(* Logix 5000 project; controller ESP_300kVA_L24ERM vendor 1 type 14 code 150 rev 33.12; software revision 33.01 *)

TASK MainTask (continuous, watchdog 500 ms) : MainProgram

MODULES
   Local : vendor 1 type 14 code 150 (Compact 0, rev 33.12)
      Discrete_IO : Embedded (Compact 1, rev 3.1, Output RPI 20 ms)
      Counters : Embedded (Compact 3, rev 1.1, Output RPI 20 ms)
      Analog_IO : Embedded (Compact 2, rev 1.1, Output RPI 80 ms)
      PowerFlex755PMM : vendor 1 type 143 code 6288 (Ethernet 192.168.2.160, rev 3.2, Output RPI 20 ms)
           PowerFlex755PMM:O.P14_DLXDINTInSP1   // Bit de Falla General
          : vendor 1 type 143 code 33184 (RhinoBP 14, rev 2.5)
          : vendor 1 type 143 code 32928 (RhinoBP 13, rev 1.1)
          : vendor 1 type 143 code 767 (RhinoBP 1, rev 2.7)
          : vendor 1 type 143 code 416 (RhinoBP 6, rev 1.8)
          : vendor 1 type 143 code 416 (RhinoBP 4, rev 1.8)
          : vendor 1 type 143 code 416 (RhinoBP 5, rev 1.8)
          : vendor 1 type 143 code 24736 (RhinoBP 7, rev 1.1)
      PowerFlex755IM : PowerFlex 755-EENET (Ethernet 192.168.2.10, rev 14.5, Output RPI 20 ms)
          : vendor 1 type 143 code 416 (RhinoBP 4, rev 1.8)
          : vendor 1 type 143 code 24736 (RhinoBP 7, rev 1.1)
          : vendor 1 type 143 code 416 (RhinoBP 5, rev 1.8)
          : vendor 1 type 143 code 767 (RhinoBP 1, rev 2.7)
          : vendor 1 type 143 code 32928 (RhinoBP 13, rev 1.1)
          : vendor 1 type 143 code 33184 (RhinoBP 14, rev 2.5)
          : vendor 1 type 143 code 416 (RhinoBP 6, rev 1.8)
END_MODULES

TYPE DIO_Fn :   // UDT Para Canales
STRUCT
   Channel : INT;   // Número del canal
   Type : BOOL;   // Typo de entrada (0:NO,1:NC) Tipo de salida (0:HA,1LA)
   Value : BOOL;   // Valor de la función
   Enable : BOOL;   // Habilitador
END_STRUCT
END_TYPE

TYPE Protecciones :
STRUCT
   Enable_HH : BOOL[32];   // Disparo por alto alto habilitado
   SetPoint_HH : REAL[32];   // Límite disparo HH
   TripTime_HH : INT[32];   // Tiempo disparo HH
   Enable_LL : BOOL[32];   // Disparo por bajo bajo habilitado
   SetPoint_LL : REAL[32];   // Límite disparo LL
   TripTime_LL : INT[32];   // Tiempo disparo LL
   Disparo_HH : BOOL[32];   // Estado de la señal de disparo HH
   Disparo_LL : BOOL[32];   // Estado de la señal de disparo LL
   Type : INT;   // Tipo de Protección
END_STRUCT
END_TYPE

ADD_ON_INSTRUCTION BMUX_16_1   (* revision 0.1 *)
// 16:1 BOOL MUX
VAR_INPUT
   INPUT : INT; {visible}   // Entrada
   SEL : INT; {visible}   // Selector
END_VAR
VAR_OUTPUT
   OUT : BOOL; {access Read Only, visible}   // Salida
END_VAR
VAR_INPUT
   TYPE : BOOL;
END_VAR
VAR
   MUX_8_1_01 : BMUX_8_1; {access None}
   MUX_8_1_02 : BMUX_8_1; {access None}
   BAND_01 : FBD_BOOLEAN_AND := (In1 := 1, In2 := 1, In3 := 1, In4 := 1, In5 := 1, In6 := 1, In7 := 1, In8 := 1); {access None}
   BAND_02 : FBD_BOOLEAN_AND := (In1 := 1, In2 := 1, In3 := 1, In4 := 1, In5 := 1, In6 := 1, In7 := 1, In8 := 1); {access None}
   BNOT_01 : FBD_BOOLEAN_NOT := (In := 1); {access None}
   BOR_01 : FBD_BOOLEAN_OR; {access None}
   __l13611DCB8D0E7587 : INT; {access None}
   __lD1E1ECCF935F20E9 : INT; {access None}
   __lCDF1D212B6E33786 : BOOL; {access None}
END_VAR

ROUTINE Logic   (* function block diagram *)
   SHEET 1
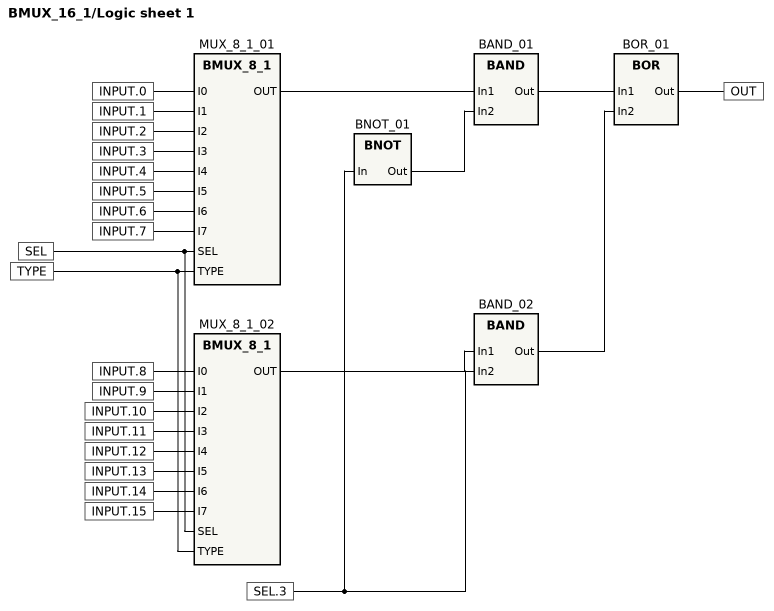
   MUX_8_1_01 : BMUX_8_1(I0 := INPUT.0, I1 := INPUT.1, I2 := INPUT.2, I3 := INPUT.3, I4 := INPUT.4, I5 := INPUT.5, I6 := INPUT.6, I7 := INPUT.7, SEL := SEL, TYPE := TYPE);
   MUX_8_1_02 : BMUX_8_1(I0 := INPUT.8, I1 := INPUT.9, I2 := INPUT.10, I3 := INPUT.11, I4 := INPUT.12, I5 := INPUT.13, I6 := INPUT.14, I7 := INPUT.15, SEL := SEL, TYPE := TYPE);
   BNOT_01 : BNOT(In := SEL.3);
   BAND_01 : BAND(In1 := MUX_8_1_01.OUT, In2 := BNOT_01.Out);
   BAND_02 : BAND(In1 := MUX_8_1_02.OUT, In2 := SEL.3);
   BOR_01 : BOR(In1 := BAND_01.Out, In2 := BAND_02.Out);
   OUT := BOR_01.Out;
END_ROUTINE
END_ADD_ON_INSTRUCTION

ADD_ON_INSTRUCTION BMUX_4_1   (* revision 0.1 *)
// 4:1 BOOL MUX
VAR_INPUT
   I0 : BOOL; {visible}   // Entrada 0
   I1 : BOOL; {visible}   // Entrada 1
   I2 : BOOL; {visible}   // Entrada 2
   I3 : BOOL; {visible}   // Entrada 3
   SEL : INT; {visible}   // Selector
END_VAR
VAR_OUTPUT
   OUT : BOOL; {visible}   // Salida
END_VAR
VAR_INPUT
   TYPE : BOOL;
END_VAR
VAR
   BAND_01 : FBD_BOOLEAN_AND := (In1 := 1, In2 := 1, In3 := 1, In4 := 1, In5 := 1, In6 := 1, In7 := 1, In8 := 1); {access None}
   BAND_02 : FBD_BOOLEAN_AND := (In1 := 1, In2 := 1, In3 := 1, In4 := 1, In5 := 1, In6 := 1, In7 := 1, In8 := 1); {access None}
   BAND_03 : FBD_BOOLEAN_AND := (In1 := 1, In2 := 1, In3 := 1, In4 := 1, In5 := 1, In6 := 1, In7 := 1, In8 := 1); {access None}
   BAND_04 : FBD_BOOLEAN_AND := (In1 := 1, In2 := 1, In3 := 1, In4 := 1, In5 := 1, In6 := 1, In7 := 1, In8 := 1); {access None}
   BOR_01 : FBD_BOOLEAN_OR; {access None}
   BNOT_01 : FBD_BOOLEAN_NOT := (In := 1); {access None}
   BNOT_02 : FBD_BOOLEAN_NOT := (In := 1); {access None}
   BAND_05 : FBD_BOOLEAN_AND := (In1 := 1, In2 := 1, In3 := 1, In4 := 1, In5 := 1, In6 := 1, In7 := 1, In8 := 1);
   BAND_06 : FBD_BOOLEAN_AND := (In1 := 1, In2 := 1, In3 := 1, In4 := 1, In5 := 1, In6 := 1, In7 := 1, In8 := 1);
   BNOT_03 : FBD_BOOLEAN_NOT := (In := 1);
   BNOT_04 : FBD_BOOLEAN_NOT := (In := 1);
   BOR_02 : FBD_BOOLEAN_OR;
   __lA34AA79BD695A9B9 : INT; {access None}
   __l3F476DF96765899A : BOOL; {access None}
   __lA5B7ACC4E5B37ACF : BOOL; {access None}
   __l435C749CB0444308 : BOOL; {access None}
   __lD1FFE671015823D2 : BOOL; {access None}
   __l62043FB7EA6F2954 : BOOL; {access None}
END_VAR

ROUTINE Logic   (* function block diagram *)
   SHEET 1
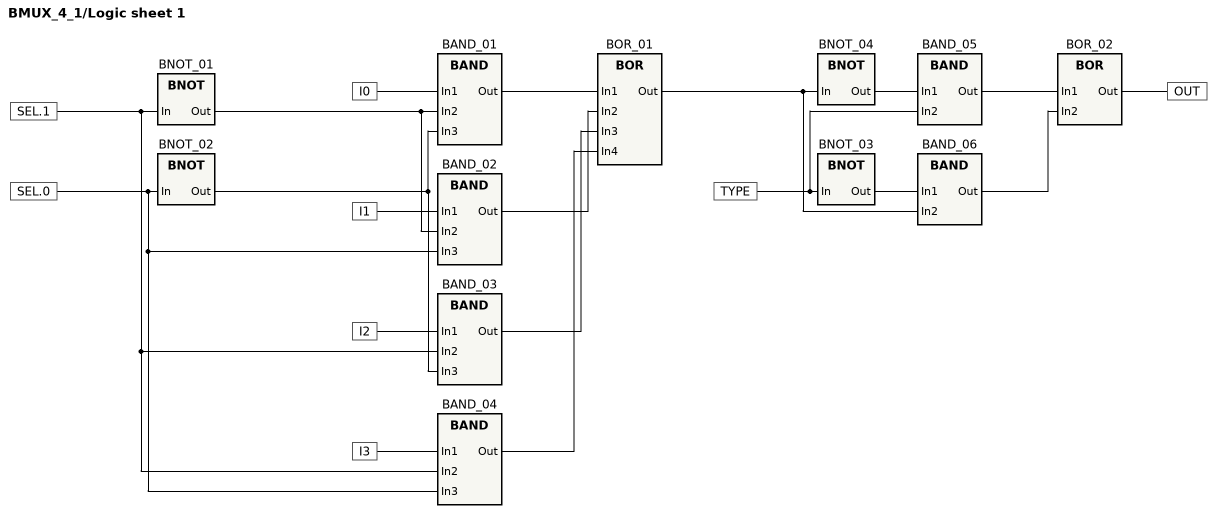
   BNOT_01 : BNOT(In := SEL.1);
   BNOT_02 : BNOT(In := SEL.0);
   BAND_01 : BAND(In1 := I0, In2 := BNOT_01.Out, In3 := BNOT_02.Out);
   BAND_02 : BAND(In1 := I1, In2 := BNOT_01.Out, In3 := SEL.0);
   BAND_03 : BAND(In1 := I2, In2 := SEL.1, In3 := BNOT_02.Out);
   BAND_04 : BAND(In1 := I3, In2 := SEL.1, In3 := SEL.0);
   BOR_01 : BOR(In1 := BAND_01.Out, In2 := BAND_02.Out, In3 := BAND_03.Out, In4 := BAND_04.Out);
   BNOT_04 : BNOT(In := BOR_01.Out);
   BNOT_03 : BNOT(In := TYPE);
   BAND_05 : BAND(In1 := BNOT_04.Out, In2 := TYPE);
   BAND_06 : BAND(In1 := BNOT_03.Out, In2 := BOR_01.Out);
   BOR_02 : BOR(In1 := BAND_05.Out, In2 := BAND_06.Out);
   OUT := BOR_02.Out;
END_ROUTINE
END_ADD_ON_INSTRUCTION

ADD_ON_INSTRUCTION BMUX_8_1   (* revision 0.1 *)
// 8:1 BOOL MUX
VAR_INPUT
   I0 : BOOL; {visible}   // Entrada 0
   I1 : BOOL; {visible}   // Entrada 1
   I2 : BOOL; {visible}   // Entrada 2
   I3 : BOOL; {visible}   // Entrada 3
   I4 : BOOL; {visible}   // Entrada 4
   I5 : BOOL; {visible}   // Entrada 5
   I6 : BOOL; {visible}   // Entrada 6
   I7 : BOOL; {visible}   // Entrada 7
   SEL : INT; {visible}   // Selector
END_VAR
VAR_OUTPUT
   OUT : BOOL; {visible}   // Salida
END_VAR
VAR_INPUT
   TYPE : BOOL;
END_VAR
VAR
   BAND_01 : FBD_BOOLEAN_AND := (In1 := 1, In2 := 1, In3 := 1, In4 := 1, In5 := 1, In6 := 1, In7 := 1, In8 := 1); {access None}
   BAND_02 : FBD_BOOLEAN_AND := (In1 := 1, In2 := 1, In3 := 1, In4 := 1, In5 := 1, In6 := 1, In7 := 1, In8 := 1); {access None}
   MUX_4_1_02 : BMUX_4_1; {access None}
   MUX_4_1_01 : BMUX_4_1; {access None}
   BNOT_01 : FBD_BOOLEAN_NOT := (In := 1); {access None}
   BOR_01 : FBD_BOOLEAN_OR; {access None}
   __l3844A21951326208 : INT; {access None}
   __l92E31AA3E07A0FB5 : BOOL; {access None}
   __lFC38970C7D342C75 : BOOL; {access None}
   __l740E29C8E41AD4FE : BOOL; {access None}
   __l47807FE8D131736A : BOOL; {access None}
   __lC8897F2B9FAED5C5 : BOOL; {access None}
   __lCFCD8E0D59ED18C9 : BOOL; {access None}
   __l6FFFD8D902218155 : BOOL; {access None}
   __lC2B98392E907BE62 : BOOL; {access None}
   __l3C983B185907781A : BOOL; {access None}
END_VAR

ROUTINE Logic   (* function block diagram *)
   SHEET 1
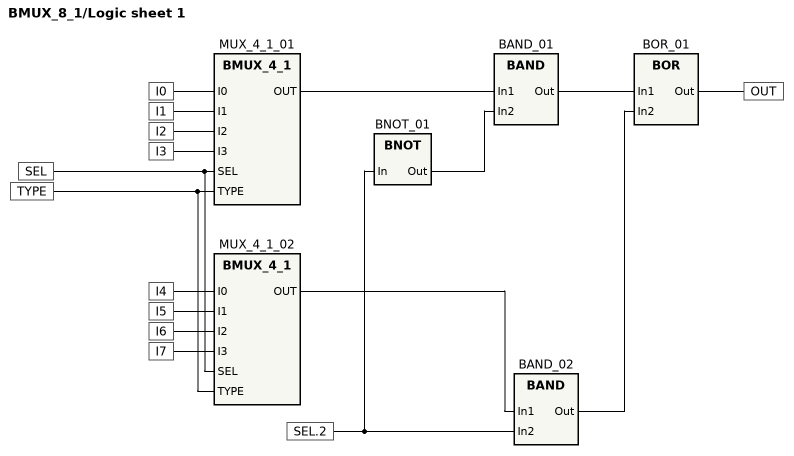
   MUX_4_1_01 : BMUX_4_1(I0 := I0, I1 := I1, I2 := I2, I3 := I3, SEL := SEL, TYPE := TYPE);
   MUX_4_1_02 : BMUX_4_1(I0 := I4, I1 := I5, I2 := I6, I3 := I7, SEL := SEL, TYPE := TYPE);
   BNOT_01 : BNOT(In := SEL.2);
   BAND_01 : BAND(In1 := MUX_4_1_01.OUT, In2 := BNOT_01.Out);
   BAND_02 : BAND(In1 := MUX_4_1_02.OUT, In2 := SEL.2);
   BOR_01 : BOR(In1 := BAND_01.Out, In2 := BAND_02.Out);
   OUT := BOR_01.Out;
END_ROUTINE
END_ADD_ON_INSTRUCTION

VAR_GLOBAL   (* controller tags *)
   ChannelSel : INT[16];
   DOChannel : INT;
   Falla_general : BOOL;
   Filtro_armonicos : BOOL;
   Reset : BOOL;
   VSD_BitFalla : DINT;
END_VAR

PROGRAM MainProgram   (* main routine MainRoutine *)
VAR
   BMUX_16_1_01 : BMUX_16_1 := (INPUT := 1743);
   BMUX_16_1_02 : BMUX_16_1 := (INPUT := 1743);
   BMUX_16_1_03 : BMUX_16_1 := (INPUT := 1743);
   BMUX_16_1_04 : BMUX_16_1 := (INPUT := 1743, TYPE := 1);
   BMUX_16_1_05 : BMUX_16_1 := (INPUT := 1743);
   BMUX_16_1_06 : BMUX_16_1 := (INPUT := 1743, SEL := 5);
   BMUX_16_1_07 : BMUX_16_1 := (INPUT := 1743, SEL := 4);
   BMUX_16_1_08 : BMUX_16_1 := (INPUT := 1743, SEL := 2, TYPE := 1);
   BMUX_16_1_09 : BMUX_16_1 := (INPUT := 1743, SEL := 3, TYPE := 1);
   BMUX_16_1_10 : BMUX_16_1 := (INPUT := 1743, SEL := 6, TYPE := 1);
   BMUX_16_1_11 : BMUX_16_1 := (INPUT := 1743, SEL := 7, TYPE := 1);
   BMUX_16_1_12 : BMUX_16_1 := (INPUT := 1743, SEL := 1, TYPE := 1);
   BMUX_16_1_13 : BMUX_16_1 := (INPUT := 1743);
   BMUX_16_1_14 : BMUX_16_1 := (INPUT := 1743);
   BMUX_16_1_15 : BMUX_16_1 := (INPUT := 1743, TYPE := 1);
   BMUX_16_1_16 : BMUX_16_1 := (INPUT := 1743);
   BMUX_16_1_17 : BMUX_16_1 := (INPUT := 1743);
   BMUX_16_1_18 : BMUX_16_1 := (INPUT := 1743, SEL := 8);
   BMUX_16_1_19 : BMUX_16_1;
   BMUX_4_1_02 : BMUX_4_1 := (SEL := 2);
   BMUX_4_1_03 : BMUX_4_1 := (SEL := 3);
   BMUX_4_1_04 : BMUX_4_1 := (SEL := 1);
   BMUX_4_1_05 : BMUX_4_1;
   BMUX_4_1_06 : BMUX_4_1;
   BMUX_4_1_07 : BMUX_4_1;
   BMUX_4_1_08 : BMUX_4_1;
   BMUX_4_1_09 : BMUX_4_1;
   BMUX_4_1_10 : BMUX_4_1;
   BMUX_4_1_11 : BMUX_4_1;
   BMUX_4_1_12 : BMUX_4_1;
   BMUX_4_1_13 : BMUX_4_1;
   BMUX_4_1_14 : BMUX_4_1;
   BMUX_4_1_15 : BMUX_4_1;
   BMUX_4_1_16 : BMUX_4_1;
   BMUX_4_1_17 : BMUX_4_1;
   BOR_01 : FBD_BOOLEAN_OR;
   BOR_02 : FBD_BOOLEAN_OR;
   BOR_03 : FBD_BOOLEAN_OR;
   BOR_04 : FBD_BOOLEAN_OR;
   BOR_05 : FBD_BOOLEAN_OR;
   BOR_06 : FBD_BOOLEAN_OR;
   BOR_07 : FBD_BOOLEAN_OR;
   BOR_08 : FBD_BOOLEAN_OR;
   BOR_09 : FBD_BOOLEAN_OR;
   BOR_10 : FBD_BOOLEAN_OR;
   BOR_11 : FBD_BOOLEAN_OR;
   BOR_12 : FBD_BOOLEAN_OR;
   BOR_13 : FBD_BOOLEAN_OR;
   BOR_14 : FBD_BOOLEAN_OR;
   BOR_15 : FBD_BOOLEAN_OR;
   BOR_16 : FBD_BOOLEAN_OR;
   BOR_17 : FBD_BOOLEAN_OR;
   BOR_18 : FBD_BOOLEAN_OR;
   BOR_19 : FBD_BOOLEAN_OR;
   BXOR_01 : FBD_BOOLEAN_XOR;
   DI_Alarma_alta_temperatura_SUT : DIO_Fn := (Channel := 4, Enable := 1);
   DI_Alarma_bajo_nivel_aceite_SUT : DIO_Fn := (Channel := 2, Type := 1, Enable := 1);
   DI_Alarma_DPS : DIO_Fn := (Channel := 7, Type := 1, Enable := 1);
   DI_Disparo_alta_presion_THP : DIO_Fn;
   DI_Disparo_alta_temperatura_filtros : DIO_Fn := (Channel := 1, Type := 1, Enable := 1);
   DI_Disparo_alta_temperatura_SUT : DIO_Fn := (Channel := 5, Enable := 1);
   DI_Disparo_alto_nivel_aceite_SUT : DIO_Fn;
   DI_Disparo_baja_presion_troncal : DIO_Fn;
   DI_Disparo_bajo_bajo_nivel_aceite_SUT : DIO_Fn := (Channel := 3, Type := 1, Enable := 1);
   DI_Disparo_puerta_abierta : DIO_Fn;
   DI_Disparo_shutdown_SCC : DIO_Fn := (Channel := 8, Enable := 1);
   DI_Disparo_sobre_tension_SUT : DIO_Fn;
   DI_Disparo_valvula_sobrepresion_SUT : DIO_Fn := (Channel := 6, Type := 1, Enable := 1);
   DI_Proteccion_termica_motor : DIO_Fn;
   DI_Reset : DIO_Fn;
   DI_Start : DIO_Fn;
   DI_Stop : DIO_Fn;
   DI_Stop_ESD : DIO_Fn := (Type := 1, Enable := 1);
   DI_Stop_ESD_Remoto : DIO_Fn;
   DO_Disparo_breaker_ESD : DIO_Fn;
   DO_Falla_general : DIO_Fn := (Channel := 2, Value := 1, Enable := 1);
   MUX_01 : MULTIPLEXER := (Status := 16#0000_0003, InstructFault := 1, SelectorInv := 1);
   Protecciones : Protecciones;
   TON_ProteccionHH : TIMER[16];
   TON_ProteccionLL : TIMER[16];
END_VAR

ROUTINE Input_Output   (* function block diagram *)
// Rutina para el control de entradas y salidas Digitales
   SHEET 1   // Funciones de entrada 1
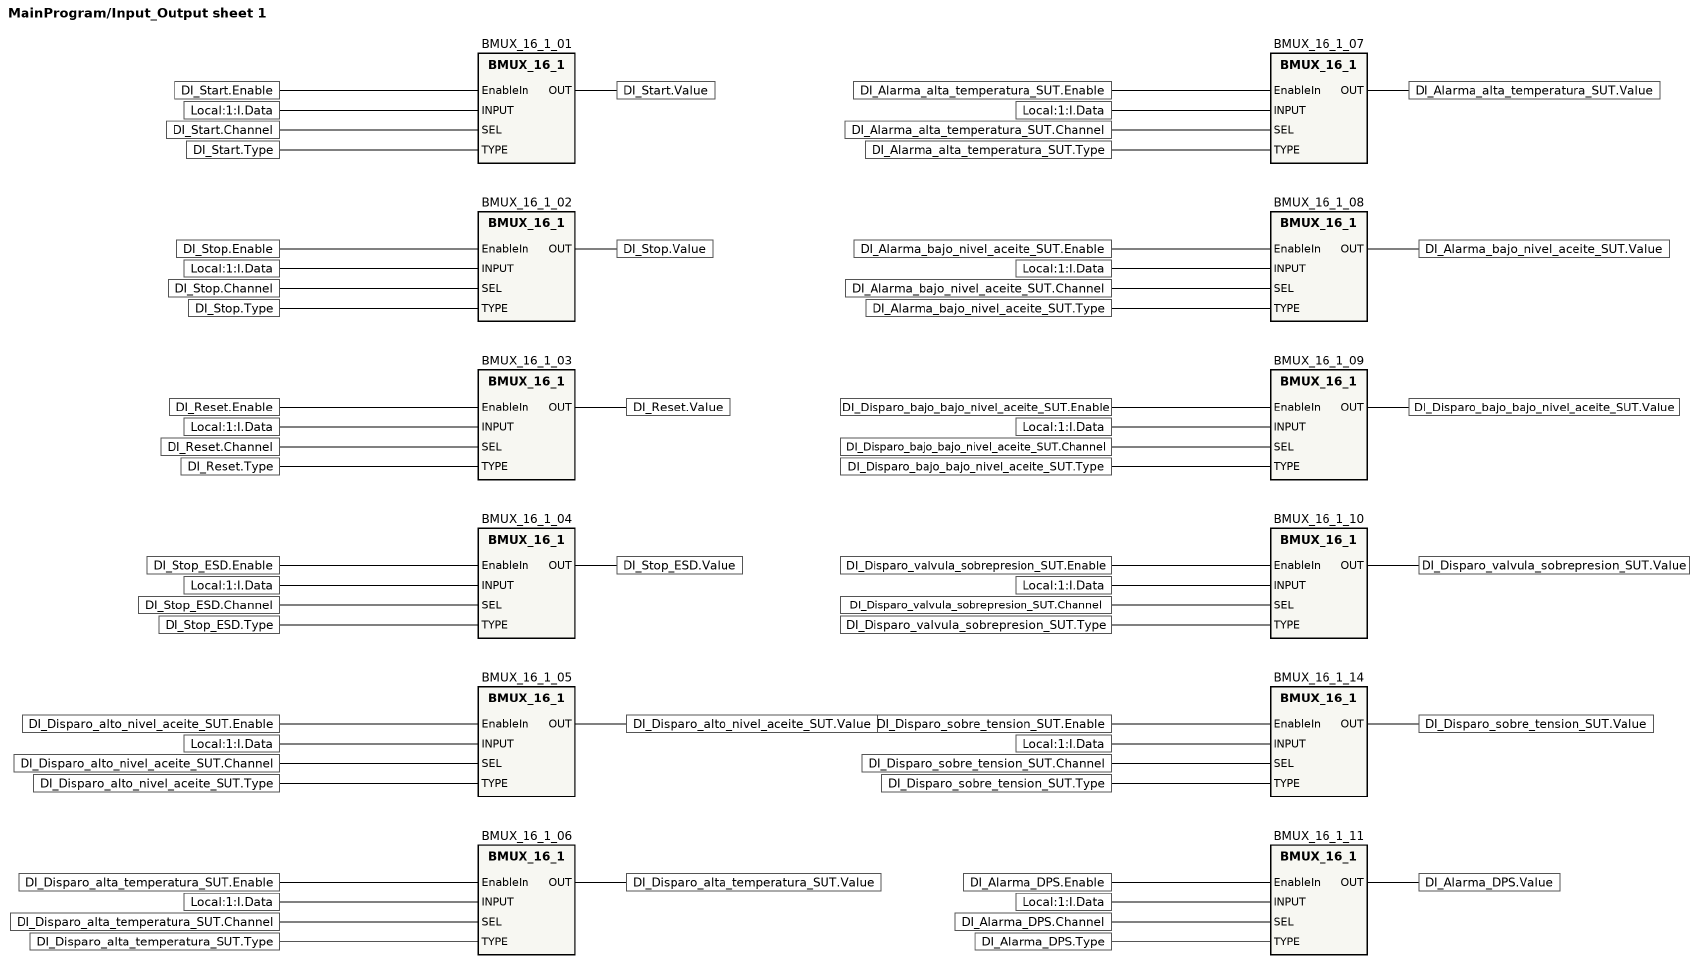
   BMUX_16_1_01 : BMUX_16_1(EnableIn := DI_Start.Enable, INPUT := Local:1:I.Data, SEL := DI_Start.Channel, TYPE := DI_Start.Type);
   BMUX_16_1_02 : BMUX_16_1(EnableIn := DI_Stop.Enable, INPUT := Local:1:I.Data, SEL := DI_Stop.Channel, TYPE := DI_Stop.Type);
   BMUX_16_1_03 : BMUX_16_1(EnableIn := DI_Reset.Enable, INPUT := Local:1:I.Data, SEL := DI_Reset.Channel, TYPE := DI_Reset.Type);
   BMUX_16_1_04 : BMUX_16_1(EnableIn := DI_Stop_ESD.Enable, INPUT := Local:1:I.Data, SEL := DI_Stop_ESD.Channel, TYPE := DI_Stop_ESD.Type);
   BMUX_16_1_05 : BMUX_16_1(EnableIn := DI_Disparo_alto_nivel_aceite_SUT.Enable, INPUT := Local:1:I.Data, SEL := DI_Disparo_alto_nivel_aceite_SUT.Channel, TYPE := DI_Disparo_alto_nivel_aceite_SUT.Type);
   BMUX_16_1_06 : BMUX_16_1(EnableIn := DI_Disparo_alta_temperatura_SUT.Enable, INPUT := Local:1:I.Data, SEL := DI_Disparo_alta_temperatura_SUT.Channel, TYPE := DI_Disparo_alta_temperatura_SUT.Type);
   DI_Start.Value := BMUX_16_1_01.OUT;
   DI_Stop.Value := BMUX_16_1_02.OUT;
   DI_Stop_ESD.Value := BMUX_16_1_04.OUT;
   DI_Reset.Value := BMUX_16_1_03.OUT;
   DI_Disparo_alto_nivel_aceite_SUT.Value := BMUX_16_1_05.OUT;
   DI_Disparo_alta_temperatura_SUT.Value := BMUX_16_1_06.OUT;
   BMUX_16_1_07 : BMUX_16_1(EnableIn := DI_Alarma_alta_temperatura_SUT.Enable, INPUT := Local:1:I.Data, SEL := DI_Alarma_alta_temperatura_SUT.Channel, TYPE := DI_Alarma_alta_temperatura_SUT.Type);
   BMUX_16_1_08 : BMUX_16_1(EnableIn := DI_Alarma_bajo_nivel_aceite_SUT.Enable, INPUT := Local:1:I.Data, SEL := DI_Alarma_bajo_nivel_aceite_SUT.Channel, TYPE := DI_Alarma_bajo_nivel_aceite_SUT.Type);
   BMUX_16_1_09 : BMUX_16_1(EnableIn := DI_Disparo_bajo_bajo_nivel_aceite_SUT.Enable, INPUT := Local:1:I.Data, SEL := DI_Disparo_bajo_bajo_nivel_aceite_SUT.Channel, TYPE := DI_Disparo_bajo_bajo_nivel_aceite_SUT.Type);
   BMUX_16_1_10 : BMUX_16_1(EnableIn := DI_Disparo_valvula_sobrepresion_SUT.Enable, INPUT := Local:1:I.Data, SEL := DI_Disparo_valvula_sobrepresion_SUT.Channel, TYPE := DI_Disparo_valvula_sobrepresion_SUT.Type);
   BMUX_16_1_14 : BMUX_16_1(EnableIn := DI_Disparo_sobre_tension_SUT.Enable, INPUT := Local:1:I.Data, SEL := DI_Disparo_sobre_tension_SUT.Channel, TYPE := DI_Disparo_sobre_tension_SUT.Type);
   BMUX_16_1_11 : BMUX_16_1(EnableIn := DI_Alarma_DPS.Enable, INPUT := Local:1:I.Data, SEL := DI_Alarma_DPS.Channel, TYPE := DI_Alarma_DPS.Type);
   DI_Alarma_alta_temperatura_SUT.Value := BMUX_16_1_07.OUT;
   DI_Disparo_bajo_bajo_nivel_aceite_SUT.Value := BMUX_16_1_09.OUT;
   DI_Alarma_bajo_nivel_aceite_SUT.Value := BMUX_16_1_08.OUT;
   DI_Disparo_valvula_sobrepresion_SUT.Value := BMUX_16_1_10.OUT;
   DI_Disparo_sobre_tension_SUT.Value := BMUX_16_1_14.OUT;
   DI_Alarma_DPS.Value := BMUX_16_1_11.OUT;
   SHEET 2   // Funciones de entrada 2
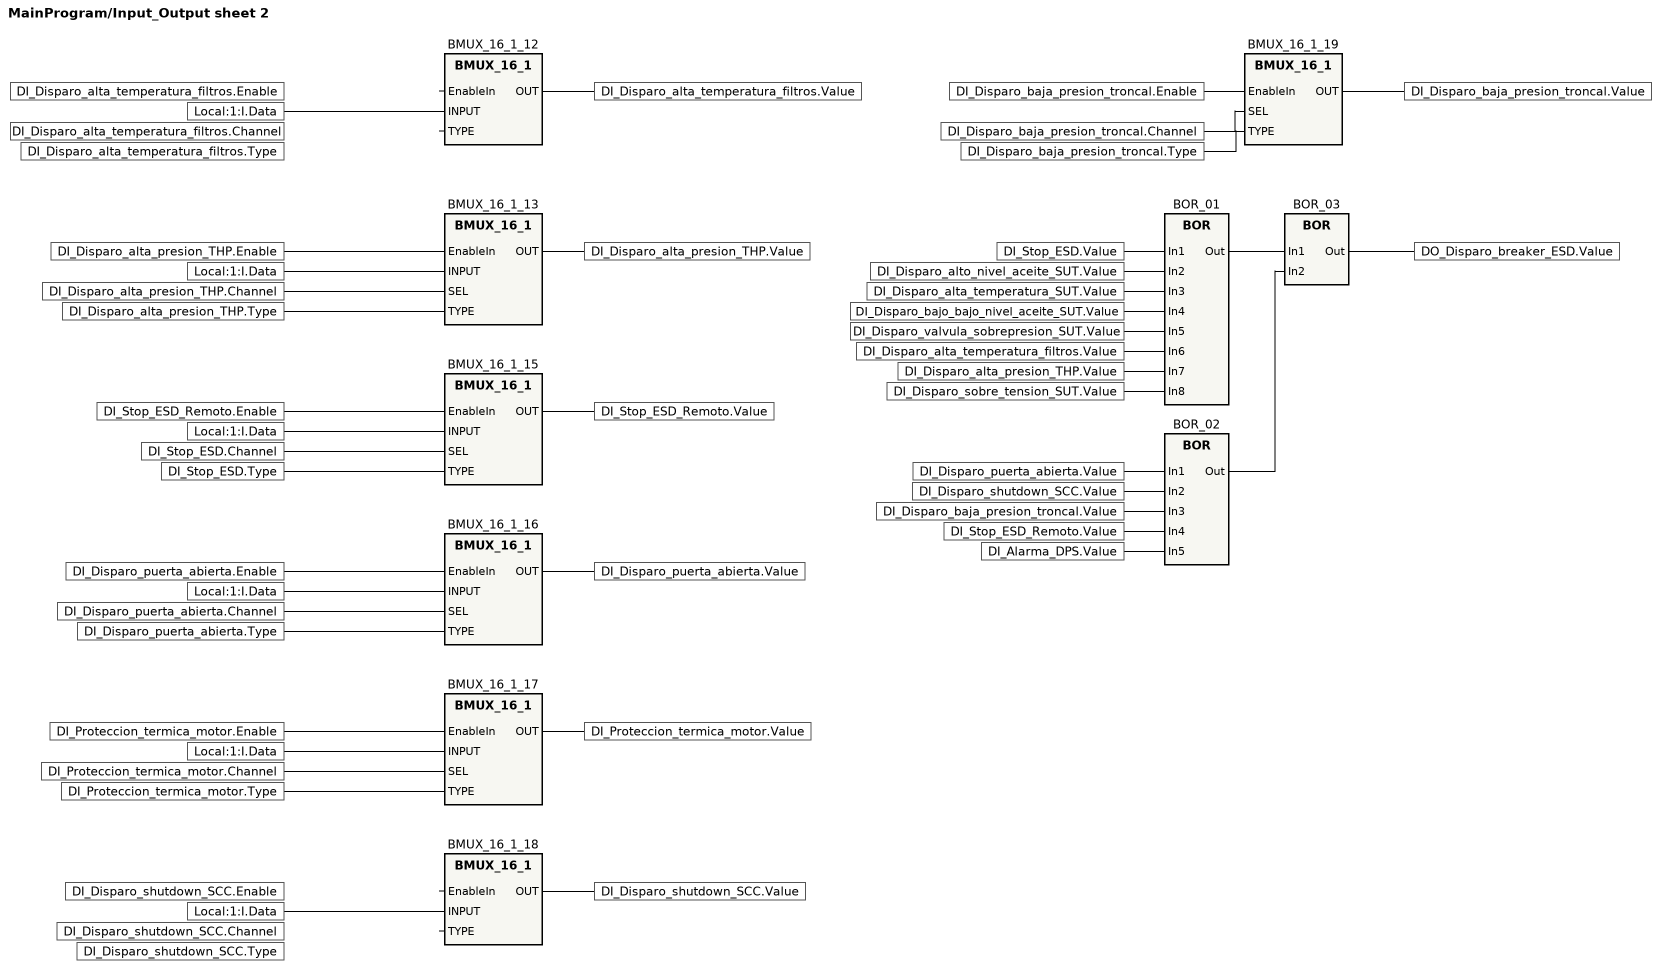
   // unwired input reference DI_Disparo_alta_temperatura_filtros.Enable
   // unwired input reference DI_Disparo_alta_temperatura_filtros.Channel
   // unwired input reference DI_Disparo_alta_temperatura_filtros.Type
   // unwired input reference DI_Disparo_shutdown_SCC.Enable
   // unwired input reference DI_Disparo_shutdown_SCC.Channel
   // unwired input reference DI_Disparo_shutdown_SCC.Type
   BMUX_16_1_12 : BMUX_16_1(INPUT := Local:1:I.Data);   // unwired pins: EnableIn TYPE
   BMUX_16_1_13 : BMUX_16_1(EnableIn := DI_Disparo_alta_presion_THP.Enable, INPUT := Local:1:I.Data, SEL := DI_Disparo_alta_presion_THP.Channel, TYPE := DI_Disparo_alta_presion_THP.Type);
   BMUX_16_1_15 : BMUX_16_1(EnableIn := DI_Stop_ESD_Remoto.Enable, INPUT := Local:1:I.Data, SEL := DI_Stop_ESD.Channel, TYPE := DI_Stop_ESD.Type);
   BMUX_16_1_16 : BMUX_16_1(EnableIn := DI_Disparo_puerta_abierta.Enable, INPUT := Local:1:I.Data, SEL := DI_Disparo_puerta_abierta.Channel, TYPE := DI_Disparo_puerta_abierta.Type);
   BMUX_16_1_17 : BMUX_16_1(EnableIn := DI_Proteccion_termica_motor.Enable, INPUT := Local:1:I.Data, SEL := DI_Proteccion_termica_motor.Channel, TYPE := DI_Proteccion_termica_motor.Type);
   BMUX_16_1_18 : BMUX_16_1(INPUT := Local:1:I.Data);   // unwired pins: EnableIn TYPE
   DI_Disparo_alta_presion_THP.Value := BMUX_16_1_13.OUT;
   DI_Proteccion_termica_motor.Value := BMUX_16_1_17.OUT;
   DI_Disparo_alta_temperatura_filtros.Value := BMUX_16_1_12.OUT;
   DI_Stop_ESD_Remoto.Value := BMUX_16_1_15.OUT;
   DI_Disparo_puerta_abierta.Value := BMUX_16_1_16.OUT;
   DI_Disparo_shutdown_SCC.Value := BMUX_16_1_18.OUT;
   BOR_01 : BOR(In1 := DI_Stop_ESD.Value, In2 := DI_Disparo_alto_nivel_aceite_SUT.Value, In3 := DI_Disparo_alta_temperatura_SUT.Value, In4 := DI_Disparo_bajo_bajo_nivel_aceite_SUT.Value, In5 := DI_Disparo_valvula_sobrepresion_SUT.Value, In6 := DI_Disparo_alta_temperatura_filtros.Value, In7 := DI_Disparo_alta_presion_THP.Value, In8 := DI_Disparo_sobre_tension_SUT.Value);
   BOR_02 : BOR(In1 := DI_Disparo_puerta_abierta.Value, In2 := DI_Disparo_shutdown_SCC.Value, In3 := DI_Disparo_baja_presion_troncal.Value, In4 := DI_Stop_ESD_Remoto.Value, In5 := DI_Alarma_DPS.Value);
   BMUX_16_1_19 : BMUX_16_1(EnableIn := DI_Disparo_baja_presion_troncal.Enable, SEL := DI_Disparo_baja_presion_troncal.Channel, TYPE := DI_Disparo_baja_presion_troncal.Type);
   BOR_03 : BOR(In1 := BOR_01.Out, In2 := BOR_02.Out);
   DI_Disparo_baja_presion_troncal.Value := BMUX_16_1_19.OUT;
   DO_Disparo_breaker_ESD.Value := BOR_03.Out;
   SHEET 3   // Salidas digitales 1
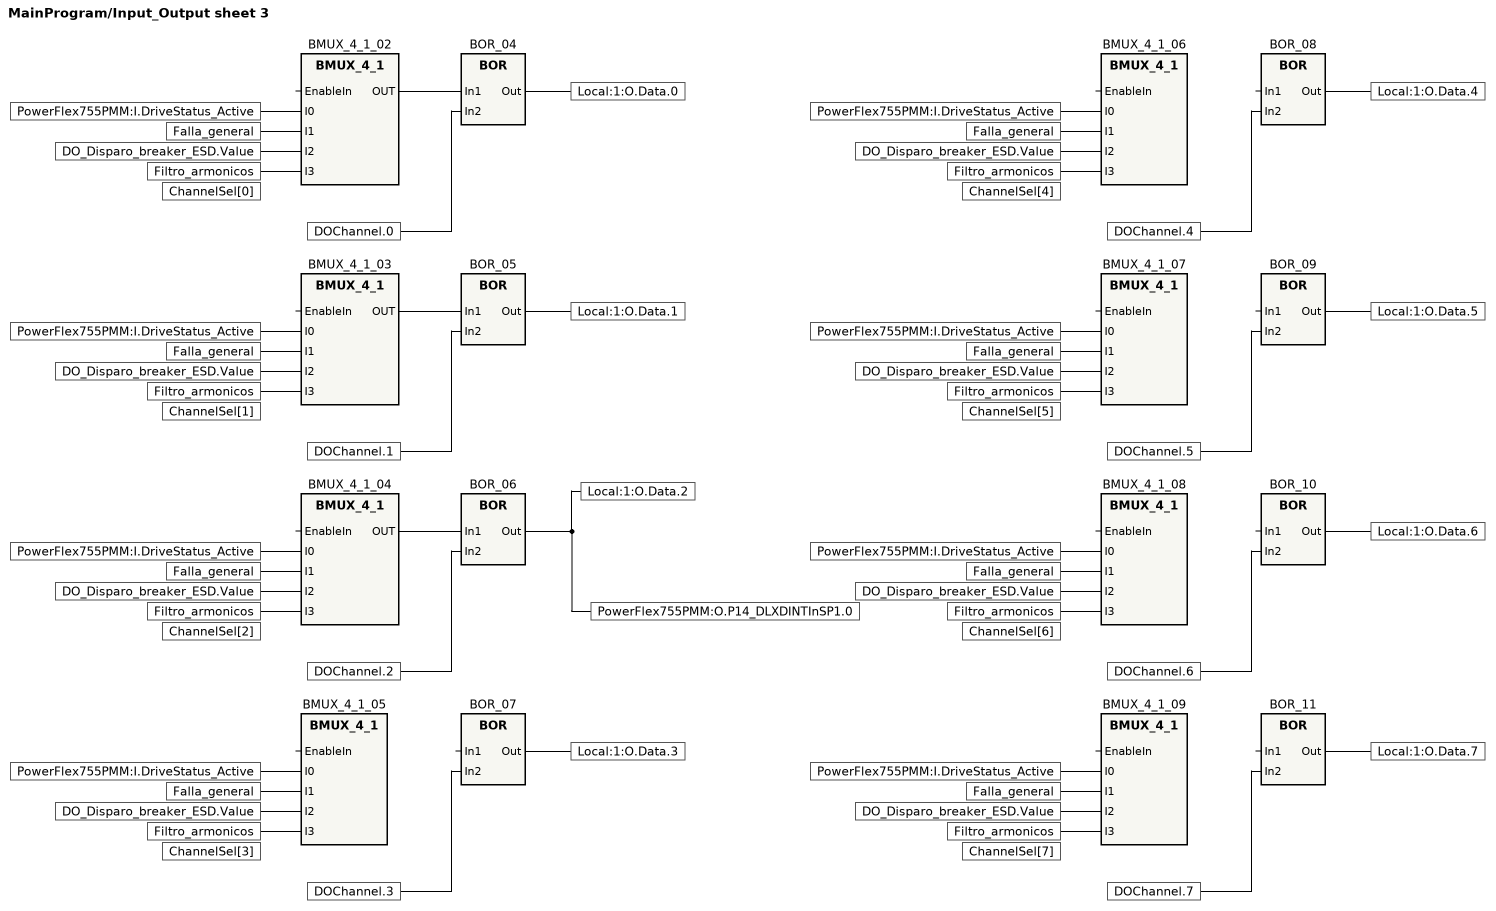
   // unwired input reference ChannelSel[0]
   // unwired input reference ChannelSel[1]
   // unwired input reference ChannelSel[2]
   // unwired input reference ChannelSel[3]
   BMUX_4_1_02 : BMUX_4_1(I0 := PowerFlex755PMM:I.DriveStatus_Active, I1 := Falla_general, I2 := DO_Disparo_breaker_ESD.Value, I3 := Filtro_armonicos);   // unwired pins: EnableIn
   BMUX_4_1_03 : BMUX_4_1(I0 := PowerFlex755PMM:I.DriveStatus_Active, I1 := Falla_general, I2 := DO_Disparo_breaker_ESD.Value, I3 := Filtro_armonicos);   // unwired pins: EnableIn
   BMUX_4_1_04 : BMUX_4_1(I0 := PowerFlex755PMM:I.DriveStatus_Active, I1 := Falla_general, I2 := DO_Disparo_breaker_ESD.Value, I3 := Filtro_armonicos);   // unwired pins: EnableIn
   BMUX_4_1_05 : BMUX_4_1(I0 := PowerFlex755PMM:I.DriveStatus_Active, I1 := Falla_general, I2 := DO_Disparo_breaker_ESD.Value, I3 := Filtro_armonicos);   // unwired pins: EnableIn
   BOR_04 : BOR(In1 := BMUX_4_1_02.OUT, In2 := DOChannel.0);
   BOR_05 : BOR(In1 := BMUX_4_1_03.OUT, In2 := DOChannel.1);
   BOR_06 : BOR(In1 := BMUX_4_1_04.OUT, In2 := DOChannel.2);
   BOR_07 : BOR(In2 := DOChannel.3);   // unwired pins: In1
   Local:1:O.Data.0 := BOR_04.Out;
   Local:1:O.Data.1 := BOR_05.Out;
   Local:1:O.Data.3 := BOR_07.Out;
   Local:1:O.Data.2 := BOR_06.Out;
   PowerFlex755PMM:O.P14_DLXDINTInSP1.0 := BOR_06.Out;
   // unwired input reference ChannelSel[4]
   // unwired input reference ChannelSel[5]
   // unwired input reference ChannelSel[6]
   // unwired input reference ChannelSel[7]
   BMUX_4_1_06 : BMUX_4_1(I0 := PowerFlex755PMM:I.DriveStatus_Active, I1 := Falla_general, I2 := DO_Disparo_breaker_ESD.Value, I3 := Filtro_armonicos);   // unwired pins: EnableIn
   BMUX_4_1_07 : BMUX_4_1(I0 := PowerFlex755PMM:I.DriveStatus_Active, I1 := Falla_general, I2 := DO_Disparo_breaker_ESD.Value, I3 := Filtro_armonicos);   // unwired pins: EnableIn
   BMUX_4_1_08 : BMUX_4_1(I0 := PowerFlex755PMM:I.DriveStatus_Active, I1 := Falla_general, I2 := DO_Disparo_breaker_ESD.Value, I3 := Filtro_armonicos);   // unwired pins: EnableIn
   BMUX_4_1_09 : BMUX_4_1(I0 := PowerFlex755PMM:I.DriveStatus_Active, I1 := Falla_general, I2 := DO_Disparo_breaker_ESD.Value, I3 := Filtro_armonicos);   // unwired pins: EnableIn
   BOR_08 : BOR(In2 := DOChannel.4);   // unwired pins: In1
   BOR_09 : BOR(In2 := DOChannel.5);   // unwired pins: In1
   BOR_10 : BOR(In2 := DOChannel.6);   // unwired pins: In1
   BOR_11 : BOR(In2 := DOChannel.7);   // unwired pins: In1
   Local:1:O.Data.4 := BOR_08.Out;
   Local:1:O.Data.5 := BOR_09.Out;
   Local:1:O.Data.6 := BOR_10.Out;
   Local:1:O.Data.7 := BOR_11.Out;
   SHEET 4   // Salidas digitales 2
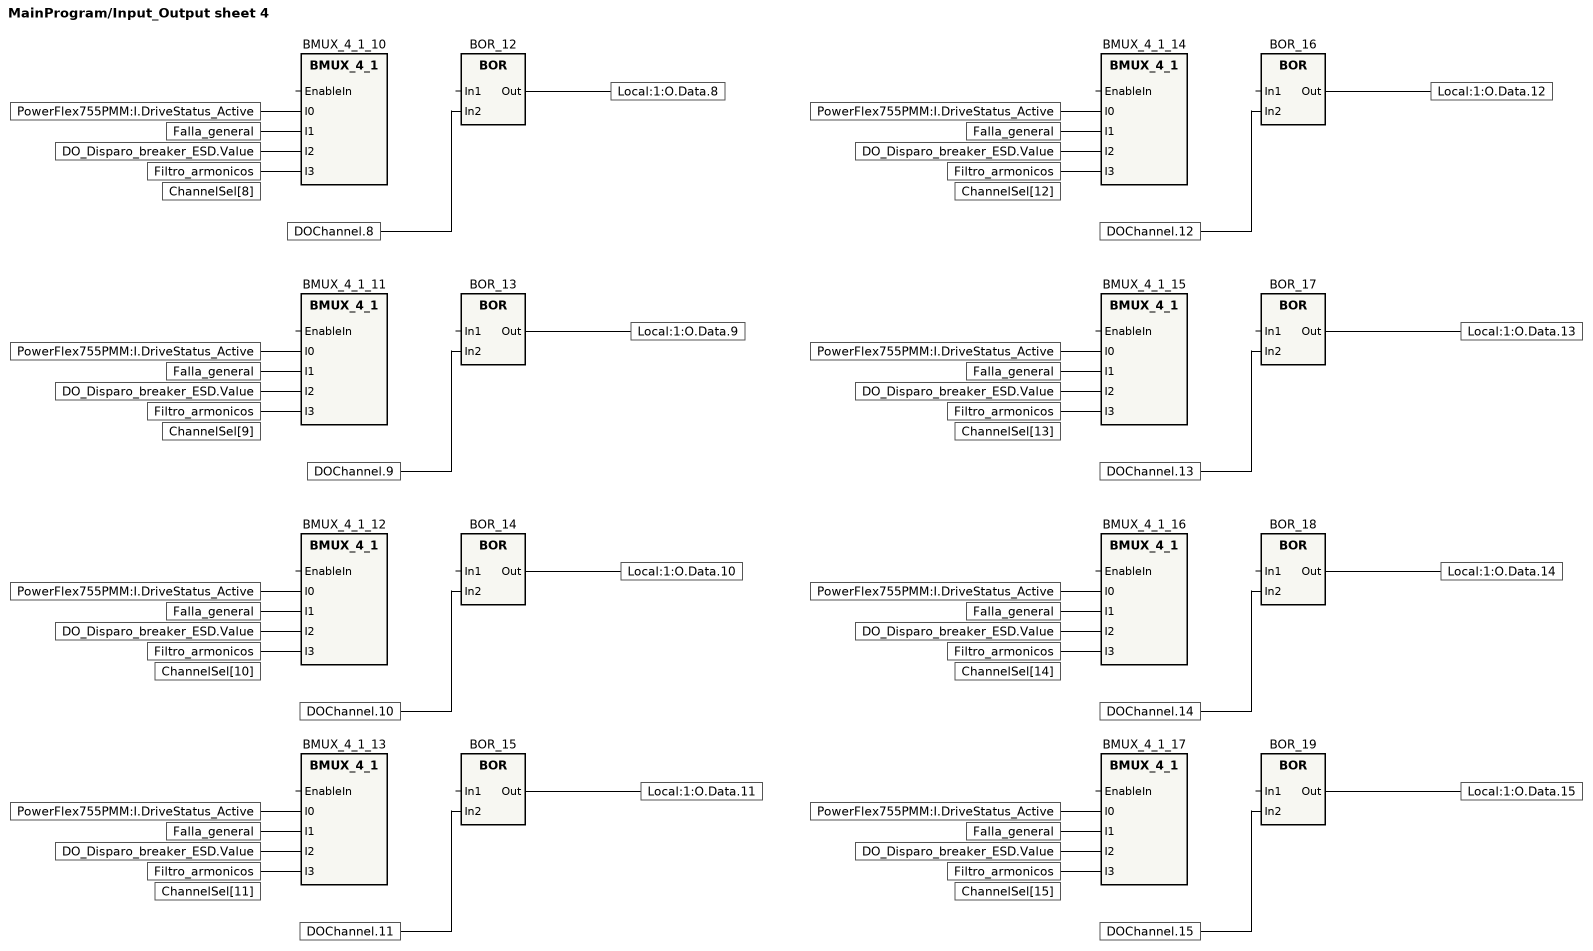
   // unwired input reference ChannelSel[8]
   // unwired input reference ChannelSel[9]
   // unwired input reference ChannelSel[10]
   // unwired input reference ChannelSel[11]
   BMUX_4_1_10 : BMUX_4_1(I0 := PowerFlex755PMM:I.DriveStatus_Active, I1 := Falla_general, I2 := DO_Disparo_breaker_ESD.Value, I3 := Filtro_armonicos);   // unwired pins: EnableIn
   BMUX_4_1_11 : BMUX_4_1(I0 := PowerFlex755PMM:I.DriveStatus_Active, I1 := Falla_general, I2 := DO_Disparo_breaker_ESD.Value, I3 := Filtro_armonicos);   // unwired pins: EnableIn
   BMUX_4_1_12 : BMUX_4_1(I0 := PowerFlex755PMM:I.DriveStatus_Active, I1 := Falla_general, I2 := DO_Disparo_breaker_ESD.Value, I3 := Filtro_armonicos);   // unwired pins: EnableIn
   BMUX_4_1_13 : BMUX_4_1(I0 := PowerFlex755PMM:I.DriveStatus_Active, I1 := Falla_general, I2 := DO_Disparo_breaker_ESD.Value, I3 := Filtro_armonicos);   // unwired pins: EnableIn
   BOR_12 : BOR(In2 := DOChannel.8);   // unwired pins: In1
   BOR_13 : BOR(In2 := DOChannel.9);   // unwired pins: In1
   BOR_14 : BOR(In2 := DOChannel.10);   // unwired pins: In1
   BOR_15 : BOR(In2 := DOChannel.11);   // unwired pins: In1
   Local:1:O.Data.8 := BOR_12.Out;
   Local:1:O.Data.10 := BOR_14.Out;
   Local:1:O.Data.9 := BOR_13.Out;
   Local:1:O.Data.11 := BOR_15.Out;
   // unwired input reference ChannelSel[12]
   // unwired input reference ChannelSel[13]
   // unwired input reference ChannelSel[14]
   // unwired input reference ChannelSel[15]
   BMUX_4_1_14 : BMUX_4_1(I0 := PowerFlex755PMM:I.DriveStatus_Active, I1 := Falla_general, I2 := DO_Disparo_breaker_ESD.Value, I3 := Filtro_armonicos);   // unwired pins: EnableIn
   BMUX_4_1_15 : BMUX_4_1(I0 := PowerFlex755PMM:I.DriveStatus_Active, I1 := Falla_general, I2 := DO_Disparo_breaker_ESD.Value, I3 := Filtro_armonicos);   // unwired pins: EnableIn
   BMUX_4_1_16 : BMUX_4_1(I0 := PowerFlex755PMM:I.DriveStatus_Active, I1 := Falla_general, I2 := DO_Disparo_breaker_ESD.Value, I3 := Filtro_armonicos);   // unwired pins: EnableIn
   BMUX_4_1_17 : BMUX_4_1(I0 := PowerFlex755PMM:I.DriveStatus_Active, I1 := Falla_general, I2 := DO_Disparo_breaker_ESD.Value, I3 := Filtro_armonicos);   // unwired pins: EnableIn
   BOR_16 : BOR(In2 := DOChannel.12);   // unwired pins: In1
   BOR_17 : BOR(In2 := DOChannel.13);   // unwired pins: In1
   BOR_18 : BOR(In2 := DOChannel.14);   // unwired pins: In1
   BOR_19 : BOR(In2 := DOChannel.15);   // unwired pins: In1
   Local:1:O.Data.12 := BOR_16.Out;
   Local:1:O.Data.14 := BOR_18.Out;
   Local:1:O.Data.13 := BOR_17.Out;
   Local:1:O.Data.15 := BOR_19.Out;
   SHEET 5   // Entradas analógicas
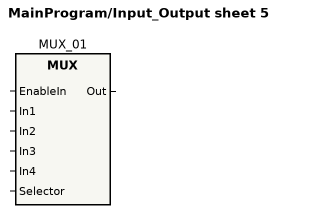
   MUX_01 : MUX();   // unwired pins: EnableIn In1 In2 In3 In4 Selector Out
END_ROUTINE

ROUTINE MainRoutine   (* ladder *)
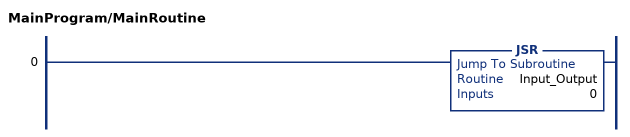
   0: JSR(Input_Output,0);
END_ROUTINE
END_PROGRAM
